INTERFACE I_VisitModules

METHOD VisitModules
VAR_INPUT
	Module : I_Module;
END_VAR
END_METHOD

END_INTERFACE

(* stored: Version 1.1.0.1, ProductVersion 3.1.4024.12
   Itf I_VisitModules: Id {4b53cfd4-bd95-4cde-b438-c14c5a9d96cb}
   Method VisitModules: Id {6d132e23-9b19-430c-b622-2d00aebe7c39} *)
